DATA_BLOCK "ID_PE_GlobalGrafcet"
{ S7_Optimized_Access := 'TRUE' }
VERSION : 0.1
NON_RETAIN
"FB_PE_GlobalGrafcet"

BEGIN

END_DATA_BLOCK

